VAR_GLOBAL
	JUnitResultFile   : JUnitResultFile<TestSuiteParameter.MaxTestSuiteCount>(TestSuiteParameter.DefaultPath);
	TestSuite		  : TestSuite<TestSuiteParameter.MaxTestCount>(ResultFile := JUnitResultFile);
	AdsLoggingEnabled : BOOL := FALSE;
END_VAR

(* stored: Version 1.1.0.1
   GVL GlobalTestSuite: Id {65860d76-d62d-4014-99f3-e31b2a55eaef} *)
